TYPE EM_Transport_WRN :
STRUCT
END_STRUCT
END_TYPE

(* stored: Version 1.1.0.1, ProductVersion 3.1.4024.12
   DUT EM_Transport_WRN: Id {3314ea2e-28cd-4578-9767-7d2555a01d3d} *)
